(* PLC project 117_1_V0.5.project, CODESYS CODESYS V3.5 SP17 Patch 3 *)
(* stored: creationDateTime 1970-01-01T00:00:00, modificationDateTime 2026-03-26T18:14:32.4070562 *)

FUNCTION_BLOCK StandLogic
  VAR_INPUT
    {attribute 'symbol' := 'none'}
    TimeManager : REFERENCE TO TimeManager;
    {attribute 'symbol' := 'none'}
    InputManager : REFERENCE TO InputManager;
    {attribute 'symbol' := 'none'}
    PIDController : REFERENCE TO BasicPIDController;
    {attribute 'symbol' := 'none'}
    ServoDriver : REFERENCE TO SM3ServoDriver;
    {attribute 'symbol' := 'none'}
    OutputManager : REFERENCE TO OutputManager;
  END_VAR
  VAR
    {attribute 'symbol' := 'none'}
    isError : BOOL := FALSE;
    {attribute 'symbol' := 'none'}
    isStateAxisOperational : BOOL := FALSE;
    {attribute 'symbol' := 'none'}
    isPowerStatus : BOOL := FALSE;
    {attribute 'symbol' := 'none'}
    isMoving : BOOL := FALSE;
    {attribute 'symbol' := 'none'}
    powerInclusionComplited : BOOL := FALSE;
    {attribute 'symbol' := 'none'}
    powerShutdownComplited : BOOL := FALSE;
    {attribute 'symbol' := 'none'}
    _controlMode : CONTROL_MODE := MANUAL;
    {attribute 'symbol' := 'none'}
    isExciterEnabled : BOOL := FALSE;
    {attribute 'symbol' := 'none'}
    isInputsReaded : BOOL;
    {attribute 'symbol' := 'none'}
    isForceRemoveLimitSwitchOn : BOOL;
    autoMoveStatus : AUTO_MOVE_STEPS := AWAIT;
    objectStatus : STATUS := NOT_COMMUNICATION;
    waitExciterOnTime : TIME := TIME#2s0ms;  (* Все что Время вкл/откл возбудителя *)
    waitExciterOffTime : TIME := TIME#2s0ms;
    cmdExciterOnOff : BOOL;  (* Команды Включение силовозбудителя *)
    cmdDisableExciter : BOOL;
    cmdPowerOn : BOOL;
    cmdPowerOff : BOOL;
    cmdErrorsReset : BOOL;
    cmdForwardJogging : BOOL;
    cmdBackwardJogging : BOOL;
    cmdChangeControlMode : BOOL;
    joggingVelocity : LREAL;  (* Ручное перемещение *)
    joggingAcceleration : LREAL;
    joggingDeceleration : LREAL;
    joggingJerk : LREAL;
    errorExciterEnableTime : BOOL;  (* Ошибки *)
    errorExciterDisableTime : BOOL;
    allErrors : ARRAY[0..15] OF BOOL;
    isInitialization : BOOL := TRUE;
    isInitialized : BOOL := FALSE;
    val : REAL;
    cc : INT;
    tenzaSensorDataArr : ARRAY[0..49] OF REAL;
    displacementSensorArr : ARRAY[0..49] OF REAL;
    nowSetpoint : REAL := 600;
    qq : BOOL;
    zz : BOOL;
    ExciterOn : SwitchingWithFeedbackControl;
    ExciterOff : SwitchingWithFeedbackControl;
    RemovingLimitSwitch : SwitchingWithFeedbackControl;
    pidStepKp : REAL;
    pidStepKi : REAL;
    pidStepKd : REAL;
    algSteps : UINT;
    stepFunction : UINT;
    diLiveCircuitsDC : BOOL;  (* Все нужные DI *)
    diFirstAlarmMushroom : BOOL;
    diSecondAlarmMushroom : BOOL;
    diLiveCircuitsAC : BOOL;
    diUpsDC_OK : BOOL;
    diUpsBattaryBad : BOOL;
    diUpsBattaryWork : BOOL;
    diUpperLimitSwitch : BOOL;
    diLowerLimitSwitch : BOOL;
    diRemovingLimitSwitch : BOOL;
    diExciter : BOOL;
    diLeftDoor : BOOL;
    diRightDoor : BOOL;
    doForcePowerLightColumn : BOOL;  (* Для поджига DO *)
    doForceRedLightColumn : BOOL;
    doForceGreenLightColumn : BOOL;
    doForceBuzzerLightColumn : BOOL;
    doForceExciter : BOOL;
    doForceRemoveLimitSwitch : BOOL;
    doStatePowerLightColumn : BOOL;  (* Состояние DO *)
    doStateRedLightColumn : BOOL;
    doStateGreenLightColumn : BOOL;
    doStateBuzzerLightColumn : BOOL;
    doStateExciter : BOOL;
    doStateRemoveLimitSwitch : BOOL;
  END_VAR

            // Чтение дискретных входов
isInputsReaded			:= _read_inputs();

// Проверка состояния силовозбудителя
isExciterEnabled		:= _check_exciter();

// Проверка состояния снятия с концевиков
isForceRemoveLimitSwitchOn := _check_removing_limit_switch();

// Проверка связи с драйвером
isStateAxisOperational	:= ServoDriver.get_axis_communication();
		
// Проверка наличия питания драйвера
isPowerStatus			:= ServoDriver.get_power_status();

IF NOT isInitialized THEN
	isInitialized := _init(TRUE);
ELSE
	// Включение и отключение дравера
	_driver_power(cmdPowerOn, cmdPowerOff);	
	
	// Режим управления
	CASE read_control_mode OF 
		MANUAL: //Ручное управление
			isMoving := _jogging(
							cmdForward 	 := cmdForwardJogging,
							cmdBackward  := cmdBackwardJogging,
							velocity	 := joggingVelocity,	
			         		acceleration := joggingAcceleration,	
			         		deceleration := joggingDeceleration,
			         		jerk		 := joggingJerk);	
							
		AUTO: // Автоматическое по алгоритму
			;
	END_CASE
	

END_IF
	














 
 IF cc >= 49 THEN
	cc := 0;
ELSE
	cc:= cc + 1;
END_IF

IF val  = 1000 THEN
	qq := TRUE;
	zz := FALSE;
ELSIF val = 0 THEN
	qq := FALSE;
	zz := TRUE;
END_IF

IF qq THEN 
		val := val - 1;
ELSIF zz THEN 
	val := val + 1;
END_IF


tenzaSensorDataArr[cc] := val;
displacementSensorArr[cc] := val + 100.0;
	

	
	//Сброс ошибок
	_reset_alarms(cmdErrorsReset);

	



	

	

	
	
	
	
	
// При аварии колонна подсвечивается красным и включается зуммер
_alarm_notification(FALSE);

// Запись статуса
objectStatus := _get_status();

// Запись выходов
_write_outputs();

          

(* Поджигает светосигнальную колонну красным *)
METHOD _alarm_notification : BOOL
  VAR_INPUT
    alarm : BOOL := FALSE;
  END_VAR
                  IF alarm THEN 
	OutputManager.set_data(varName := outRedLightColumn,	enable := TRUE);
	OutputManager.set_data(varName := outBuzzerLightColumn, enable := TRUE);
ELSE
	OutputManager.set_data(varName := outRedLightColumn,	enable := FALSE);
	OutputManager.set_data(varName := outBuzzerLightColumn, enable := FALSE);
END_IF
                
END_METHOD
END_FUNCTION_BLOCK
